(*
SPDX-FileCopyrightText: © 2026 Oleksandr Tiutyk <trofimich@gmail.com>
SPDX-License-Identifier: MIT
License: https://opensource.org/license/mit
*)

{attribute 'no_explicit_call' := 'do not call this function block directly'} 
FUNCTION_BLOCK SimpleEvent EXTENDS Event IMPLEMENTS INamed
VAR
	{attribute 'hide'} 
	_ClassName : STRING := __POUNAME();

	{attribute 'hide'} 
	_Name : WSTRING;
END_VAR

{attribute 'monitoring' := 'call'}
PROPERTY ClassName : REFERENCE TO STRING
GET
ClassName REF= _ClassName;
END_GET
END_PROPERTY

//!<param name="bInitRetains">if TRUE, the retain variables are initialized (warm start / cold start)</param>

//!<param name="bInCopyCode">if TRUE, the instance afterwards gets moved into the copy code (online change)</param>

METHOD FB_init : BOOL
VAR_INPUT
	
	bInitRetains	: BOOL;
	
	bInCopyCode	: BOOL;
	sourceObject : IObject := 0;
	name : WSTRING := "";
END_VAR
_Name := name;
END_METHOD

{attribute 'monitoring' := 'call'}
PROPERTY FINAL Name : REFERENCE TO WSTRING
GET
Name REF= _Name;
END_GET
END_PROPERTY

{attribute 'monitoring' := 'call'}
PROPERTY NamespaceName : REFERENCE TO STRING
GET
NamespaceName REF= CurrentNamespace.Name;
END_GET
END_PROPERTY

{attribute 'monitoring' := 'call'}
PROPERTY SelfSize : ULINT
GET
SelfSize := XSIZEOF(THIS^);
END_GET
END_PROPERTY

END_FUNCTION_BLOCK

(* stored: Version 1.1.0.1
   POU SimpleEvent: Id {6068111a-5f7a-4513-bc9f-2ae69d62cec9}, SpecialFunc None
   Property ClassName: Id {74c80bc7-04ea-415b-b755-fddcf5a7aecd}
   Get Get: Id {0b51e612-0055-4cf8-b992-12a817738a31}
   Method FB_init: Id {95fe79f8-57ab-4f8f-8458-df22c083e6ed}
   Property Name: Id {4cc1da98-6df4-40c6-a0ac-2b058bef2a45}
   Get Get: Id {ad2c60a7-000d-4095-a6d7-745948b89b90}
   Property NamespaceName: Id {1b34e43a-b41f-4a0e-a898-2b2522bb7be9}
   Get Get: Id {3f60aa11-e0bd-4b9d-855a-97e19aaee39b}
   Property SelfSize: Id {f60f572d-0842-4bee-822f-fb69e5ace254}
   Get Get: Id {45257b9e-307e-4ab0-ac78-b362d5465874} *)
